// TIA Portal project "hwPulito_V18" (V18)

(* hardware
DEVICE "S71500/ET200MP station_1"  S7-1500 station
   slot 0: "Telaio di montaggio_0"  Rack  6ES7 590-1***0-0AA0
   slot 1: "PLC_1"  CPU 1516-3 PN/DP  6ES7 516-3AN01-0AB0  V1.8
      slot 3: "Display CPU_1"  6ES7591-1BA00-0AA0
   slot 2: "DI 32x24VDC HF_1"  DI 32x24VDC HF  6ES7 521-1BL00-0AB0  V1.0
   slot 3: "DQ 32x24VDC/0.5A HF_1"  DQ 32x24VDC/0.5A HF  6ES7 522-1BL01-0AB0  V1.0
   slot 4: "AI 8xU/I/RTD/TC ST_1"  AI 8xU/I/RTD/TC ST  6ES7 531-7KF00-0AB0  V1.0
   slot 5: "AQ 4xU/I ST_1"  AQ 4xU/I ST  6ES7 532-5HD00-0AB0  V1.0
*)

// ===== PLC "PLC_1"  CPU 1516-3 PN/DP =====

ORGANIZATION_BLOCK "Main"   // OB1, LAD, ProgramCycle
TITLE = "Main Program Sweep (Cycle)"
{ S7_Optimized_Access := 'TRUE' }
VERSION : 0.1
   VAR_INPUT
      Initial_Call : Bool;   // Initial call of this OB
      Remanence : Bool;   // =True, if remanent data are available
   END_VAR
BEGIN
END_ORGANIZATION_BLOCK